TYPE ST_ELM3xxxPAIInfoData :
STRUCT
	nCPU_Usage: UINT;
	nDeviceState: UINT;
	nOperating_Time: UDINT;
	nOverTemperature_Time: UDINT;
	fDeviceTemperature: REAL;
	fDeviceTemperatureMin: REAL;
	fDeviceTemperatureMax: REAL;
END_STRUCT
END_TYPE

(* stored: Version 1.1.0.1, ProductVersion 3.1.4024.12
   DUT ST_ELM3xxxPAIInfoData: Id {4d476d36-6167-47d5-94e9-c3fe0b9ca817} *)
